INTERFACE I_ValueWriter

METHOD ABSTRACT ValueWriter : HRESULT
VAR_IN_OUT
    stCtx  : ST_WriteContext;
END_VAR
VAR_INPUT
    anyIn : T_ANY;
END_VAR
END_METHOD

END_INTERFACE

(* stored: Version 1.1.0.1
   Itf I_ValueWriter: Id {cb53fd15-1bee-4271-bef3-792cb4a22e72}
   Method ValueWriter: Id {79795000-1c35-41ae-8483-d11fc25b9e78} *)
